// TIA Portal V16 export
// export: Created 2021-09-08T12:46:07.0976159Z, ExportSetting WithDefaults, DisplayName Totally Integrated Automation Portal, DisplayVersion V16 Update 3, DisplayName TIA Portal Version Control Interface, DisplayVersion V16 Update 2, DisplayName TIA Portal Openness, DisplayVersion V16 Update 3, DisplayName TIA Portal Teamcenter Gateway, DisplayVersion V16, DisplayName STEP 7 Professional, DisplayVersion V16 Update 3, DisplayName STEP 7 Safety, DisplayVersion V16, DisplayName WinCC Advanced, DisplayVersion V16 Update 3
ORGANIZATION_BLOCK "Cyclic interrupt"   // OB30, LAD, CyclicInterrupt
{ S7_Optimized_Access := 'TRUE' }
VERSION : 0.1
// stored: AutoNumber true, IsIECCheckEnabled false, SetENOAutomatically false
   VAR_INPUT
      Initial_Call : Bool;   // Initial call of this OB
      Event_Count : Int;   // Events discarded
   END_VAR
BEGIN

REGION Network 1: Plc analogs
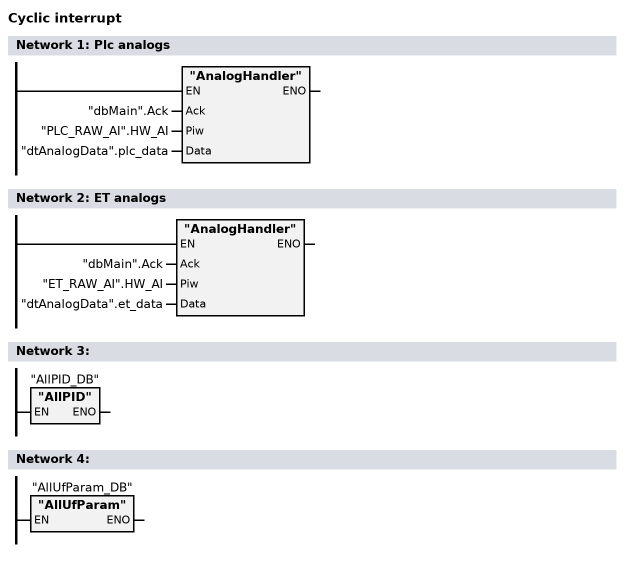
   RUNG wire#powerrail
      "AnalogHandler"(Ack := "dbMain".Ack, Piw := "PLC_RAW_AI".HW_AI, Data := "dtAnalogData".plc_data)
   END_RUNG
   // the same network as SCL:
   "AnalogHandler"(Ack := "dbMain".Ack, Piw := "PLC_RAW_AI".HW_AI, Data := "dtAnalogData".plc_data);
END_REGION

REGION Network 2: ET analogs
   RUNG wire#powerrail
      "AnalogHandler"(Ack := "dbMain".Ack, Piw := "ET_RAW_AI".HW_AI, Data := "dtAnalogData".et_data)
   END_RUNG
   // the same network as SCL:
   "AnalogHandler"(Ack := "dbMain".Ack, Piw := "ET_RAW_AI".HW_AI, Data := "dtAnalogData".et_data);
END_REGION

REGION Network 3
   RUNG wire#powerrail
      "AllPID_DB"()
   END_RUNG
   // the same network as SCL:
   "AllPID_DB"();   // "AllPID"
END_REGION

REGION Network 4
   RUNG wire#powerrail
      "AllUfParam_DB"()
   END_RUNG
   // the same network as SCL:
   "AllUfParam_DB"();   // "AllUfParam"
END_REGION
END_ORGANIZATION_BLOCK
